(* Logix 5000 project; controller STAT 1756-L72 rev 20.12; software revision 20.04; part 11 of 34 *)
(* tags used below, declared in another part *)
   ai_flow_L1 : REAL;
   ai_flow_L2 : REAL;
   ai_flow_L3 : REAL;
   aux2_P1 : BOOL;
   AUX2_P2 : BOOL;
   aux_P1_ETANG : BOOL;
   AUX_P2 : BOOL;
   AUX_P5_RINC : BOOL;
   B10 : DINT[20];
   B14 : DINT[30];
   B16 : DINT[30];
   B17 : DINT[30];
   B3 : DINT[256];
   B9 : DINT[40];
   EAU_VILLE : BOOL;
   F8 : REAL[256];
   I19_000_Bit14 : ALIAS FOR I19[0].14;   // vanne eau ville open
   I19_000_Bit15 : ALIAS FOR I19[0].15;   // vanne eau ville closed
   I19_001_Bit00 : ALIAS FOR I19[1].0;   // pulse eau de ville
   I1_005_Bit15 : ALIAS FOR I1[5].15;
   I1_008_Bit01 : ALIAS FOR I1[8].1;   // Hand Automaat stormbekken
   I1_008_Bit02 : ALIAS FOR I1[8].2;   // Start pomp 1 stormbekken
   I1_008_Bit03 : ALIAS FOR I1[8].3;   // Stop pomp 1 stormbekken
   I1_008_Bit04 : ALIAS FOR I1[8].4;   // Start pomp 2 stormbekken
   I1_008_Bit05 : ALIAS FOR I1[8].5;   // Stop pomp 2 stormbekken
   I1_008_Bit06 : ALIAS FOR I1[8].6;   // Start P3 stormbekken
   I1_008_Bit07 : ALIAS FOR I1[8].7;   // Stop P3 stormbekken
   I1_008_Bit08 : ALIAS FOR I1[8].8;   // Start PD1 Biocide
   I1_008_Bit09 : ALIAS FOR I1[8].9;   // Stop PD1 biocide
   I1_008_Bit10 : ALIAS FOR I1[8].10;   // start pd2 biocide
   I1_008_Bit11 : ALIAS FOR I1[8].11;   // stop pd2 biocide
   I1_009_Bit05 : ALIAS FOR I1[9].5;   // Pomp 1 in driehoek
   I1_009_Bit06 : ALIAS FOR I1[9].6;   // Pomp 1 in ster
   I1_009_Bit09 : ALIAS FOR I1[9].9;   // Pomp 2 in driehoek
   I1_009_Bit10 : ALIAS FOR I1[9].10;   // Pomp 2 in ster
   I1_009_Bit13 : ALIAS FOR I1[9].13;   // Pomp 3 in driehoek
   I1_009_Bit14 : ALIAS FOR I1[9].14;   // Pomp 3 in ster
   I1_010_Bit05 : ALIAS FOR I1[10].5;   // Vlotterschak lal stormbekken
   I1_010_Bit07 : ALIAS FOR I1[10].7;   // Inpuls promag 33 debiet
   I1_010_Bit10 : ALIAS FOR I1[10].10;   // Noodstop relais ok stormbekken
   I26_000 : ALIAS FOR I26[0];
   I26_003 : ALIAS FOR I26[3];
   I26_004 : ALIAS FOR I26[4];
   I26_005 : ALIAS FOR I26[5];
   I26_007 : ALIAS FOR I26[7];
   I28_000 : ALIAS FOR I28[0];
   I28_001 : ALIAS FOR I28[1];
   I28_002 : ALIAS FOR I28[2];
   I2_000_Bit04 : ALIAS FOR I2[0].4;   // Deelnoodstop cl6 eurowater
   I2_000_Bit05 : ALIAS FOR I2[0].5;   // Deelnoodstop cl7 IBT A
   I4_000_Bit02 : ALIAS FOR I4[0].2;   // defaut drive P4
   I5_001_Bit12 : ALIAS FOR I5[1].12;   // EV6_OPEN
   I5_001_Bit13 : ALIAS FOR I5[1].13;   // EV6_TOE
   I5_001_Bit14 : ALIAS FOR I5[1].14;   // EV7_TOE
   I6_000_Bit00 : ALIAS FOR I6[0].0;   // totaal debiet tfb1
   I6_000_Bit01 : ALIAS FOR I6[0].1;   // totaal debiet stfa 2
   I6_000_Bit07 : ALIAS FOR I6[0].7;   // pulsteller debiet ontijzer 2
   I6_000_Bit15 : ALIAS FOR I6[0].15;   // Lus 1 niveau reservoir kontakt 3
   I6_001_Bit00 : ALIAS FOR I6[1].0;   // hoog alarm ketel pretraitec water
   I6_001_Bit01 : ALIAS FOR I6[1].1;   // Lus 1 niveau ketel hoog
   I6_001_Bit02 : ALIAS FOR I6[1].2;   // laag alarm pretraitec water
   I6_001_Bit03 : ALIAS FOR I6[1].3;   // zeer laag alarm pretraitec water
   I6_001_Bit05 : ALIAS FOR I6[1].5;   // debietsmeting q2 pulsen
   I6_001_Bit08 : ALIAS FOR I6[1].8;   // debietsmeting q3 pulsen
   I7_000_Bit07 : ALIAS FOR I7[0].7;   // hoog alarm ketel tampon
   I7_001_Bit07 : ALIAS FOR I7[1].7;   // q4 inpulsen osmose globaal
   I8_000_Bit04 : ALIAS FOR I8[0].4;   // niveau kuip 20m hoog alarm
   I8_001_Bit09 : ALIAS FOR I8[1].9;   // Schakelaar hand autom cl6
   I9_000_Bit06 : ALIAS FOR I9[0].6;   // Drukknop start CL6 S1
   I9_000_Bit07 : ALIAS FOR I9[0].7;   // Drukknop stop CL6 S1
   I9_000_Bit09 : ALIAS FOR I9[0].9;   // Hand_Auto CL7
   I9_000_Bit10 : ALIAS FOR I9[0].10;   // Drukknop start CL7 P3
   I9_000_Bit11 : ALIAS FOR I9[0].11;   // Drukknop stop CL7 P3
   I9_000_Bit14 : ALIAS FOR I9[0].14;   // Drukknop start CL7 P5
   I9_000_Bit15 : ALIAS FOR I9[0].15;   // Drukknop stop CL7 P5
   ibtlancy1 : DINT;
   KRK_K2 : DINT;
   L1_stat : DINT[20];
   LDN_L2 : REAL;
   LDN_L3 : REAL;
   mem1 : REAL;
   mem3 : REAL;
   mem_water_flow_to_l1 : REAL;
   mem_water_flow_to_l2 : REAL;
   mem_water_flow_to_l31 : REAL;
   MW : BOOL;
   N11 : DINT[150];
   N12 : DINT[230];
   N12_219 : REAL;
   N12_220 : REAL;
   N12_221 : REAL;
   N13 : DINT[230];
   N24 : DINT[80];
   O13_001_Bit13 : ALIAS FOR O13[1].13;   // vanne eau de ville
   O15_001_Bit10 : ALIAS FOR O15[1].10;   // EV6 EV6
   O1_011_Bit00 : ALIAS FOR O1[11].0;
   O1_011_Bit01 : ALIAS FOR O1[11].1;
   O1_011_Bit02 : ALIAS FOR O1[11].2;
   O1_011_Bit03 : ALIAS FOR O1[11].3;
   O1_011_Bit04 : ALIAS FOR O1[11].4;
   O1_011_Bit05 : ALIAS FOR O1[11].5;
   O1_011_Bit06 : ALIAS FOR O1[11].6;
   O1_011_Bit07 : ALIAS FOR O1[11].7;
   O1_011_Bit08 : ALIAS FOR O1[11].8;
   O1_011_Bit09 : ALIAS FOR O1[11].9;
   O1_011_Bit10 : ALIAS FOR O1[11].10;
   ons7 : BOOL;
   ons8 : BOOL;
   ons9 : BOOL;
   P1_ETANG : BOOL;
   P2_ETANG : BOOL;
   P3 : BOOL;
   P4 : BOOL;
   P5_regen : BOOL;
   PRES_LIGNE : REAL;
   QUAT_Q2 : REAL;
   S1 : BOOL;
   s_bp_wissel_P2_usi_tfb : BOOL;   // choix p2 etang vers tfb (1) ou usine (0)
   S_LVL_VIJVER : REAL;
   scp_KRK2 : SCP;
   scp_l1_flow : SCP;
   scp_l2_flow : SCP;
   scp_l3_flow : SCP;
   scp_LDN_2 : SCP;
   scp_LDN_3 : SCP;
   scp_N12_219 : SCP;
   scp_N12_220 : SCP;
   scp_N12_221 : SCP;
   scp_PRES_LIGNE : SCP;
   scp_quat_2 : SCP;
   t1min : TIMER;
   T27 : TIMER[100];
   T4 : TIMER[200];
   water_flow_to_l1 : REAL;
   water_flow_to_l1_inst : REAL;
   water_flow_to_l2 : REAL;
   water_flow_to_l2_inst : REAL;
   water_flow_to_l3 : REAL;
   water_flow_to_l3_inst1 : REAL;
(* ibt, continued *)

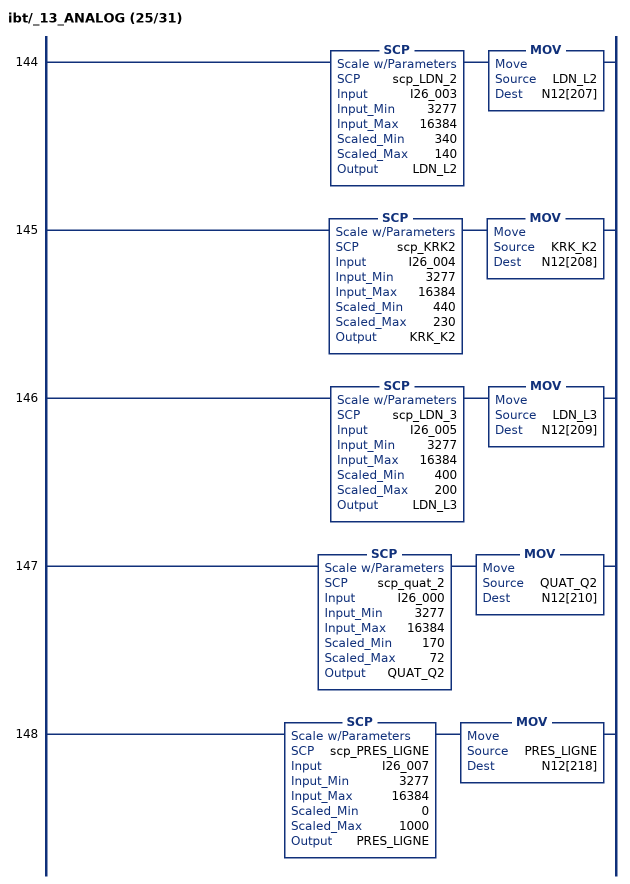
   [picture p154: ibt/_13_ANALOG rungs 144-148]
   144: SCP(scp_LDN_2,I26_003,3277,16384,340,140,LDN_L2)MOV(LDN_L2,N12[207]);
   145: SCP(scp_KRK2,I26_004,3277,16384,440,230,KRK_K2)MOV(KRK_K2,N12[208]);
   146: SCP(scp_LDN_3,I26_005,3277,16384,400,200,LDN_L3)MOV(LDN_L3,N12[209]);
   147: SCP(scp_quat_2,I26_000,3277,16384,170,72,QUAT_Q2)MOV(QUAT_Q2,N12[210]);
   148: SCP(scp_PRES_LIGNE,I26_007,3277,16384,0,1000,PRES_LIGNE)MOV(PRES_LIGNE,N12[218]);
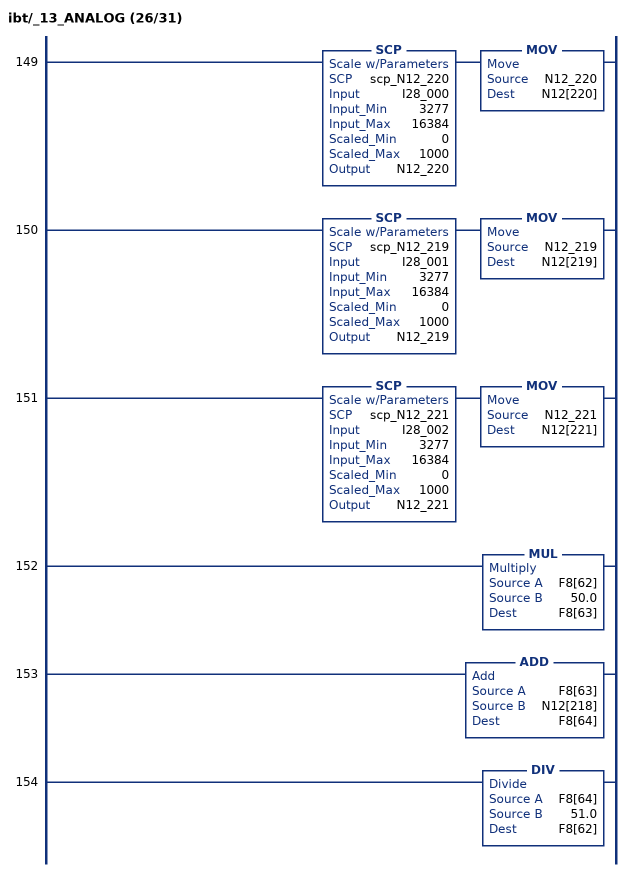
   149: SCP(scp_N12_220,I28_000,3277,16384,0,1000,N12_220)MOV(N12_220,N12[220]);
   150: SCP(scp_N12_219,I28_001,3277,16384,0,1000,N12_219)MOV(N12_219,N12[219]);
   151: SCP(scp_N12_221,I28_002,3277,16384,0,1000,N12_221)MOV(N12_221,N12[221]);
   152: MUL(F8[62],50.0,F8[63]);
   153: ADD(F8[63],N12[218],F8[64]);
   154: DIV(F8[64],51.0,F8[62]);
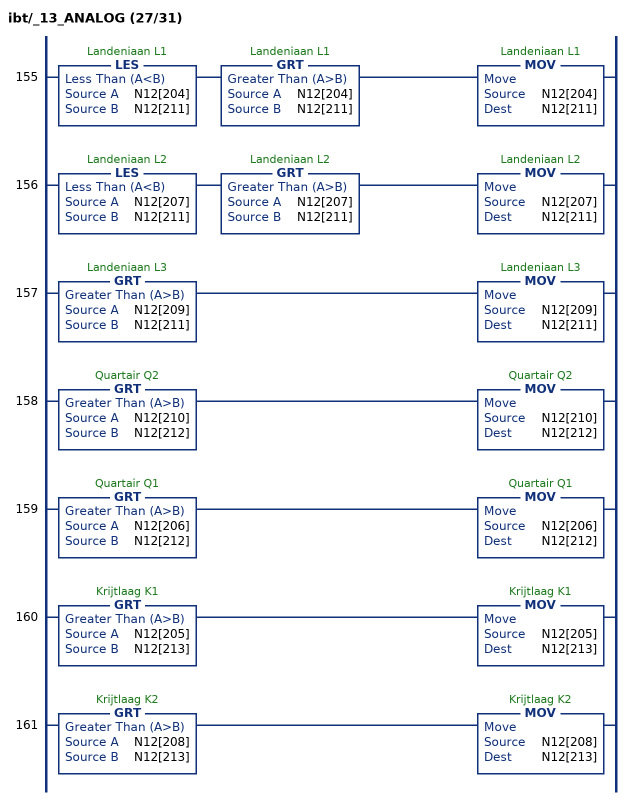
   155: LES(N12[204],N12[211])GRT(N12[204],N12[211])MOV(N12[204],N12[211]);
   156: LES(N12[207],N12[211])GRT(N12[207],N12[211])MOV(N12[207],N12[211]);
   157: GRT(N12[209],N12[211])MOV(N12[209],N12[211]);
   158: GRT(N12[210],N12[212])MOV(N12[210],N12[212]);
   159: GRT(N12[206],N12[212])MOV(N12[206],N12[212]);
   160: GRT(N12[205],N12[213])MOV(N12[205],N12[213]);
   161: GRT(N12[208],N12[213])MOV(N12[208],N12[213]);
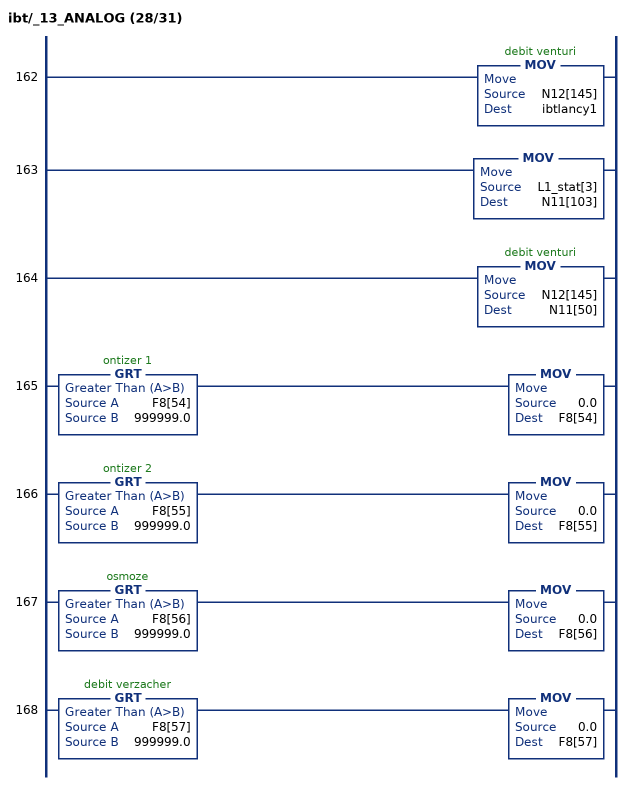
   162: MOV(N12[145],ibtlancy1);
   163: MOV(L1_stat[3],N11[103]);
   164: MOV(N12[145],N11[50]);
   165: GRT(F8[54],999999.0)MOV(0.0,F8[54]);
   166: GRT(F8[55],999999.0)MOV(0.0,F8[55]);
   167: GRT(F8[56],999999.0)MOV(0.0,F8[56]);
   168: GRT(F8[57],999999.0)MOV(0.0,F8[57]);
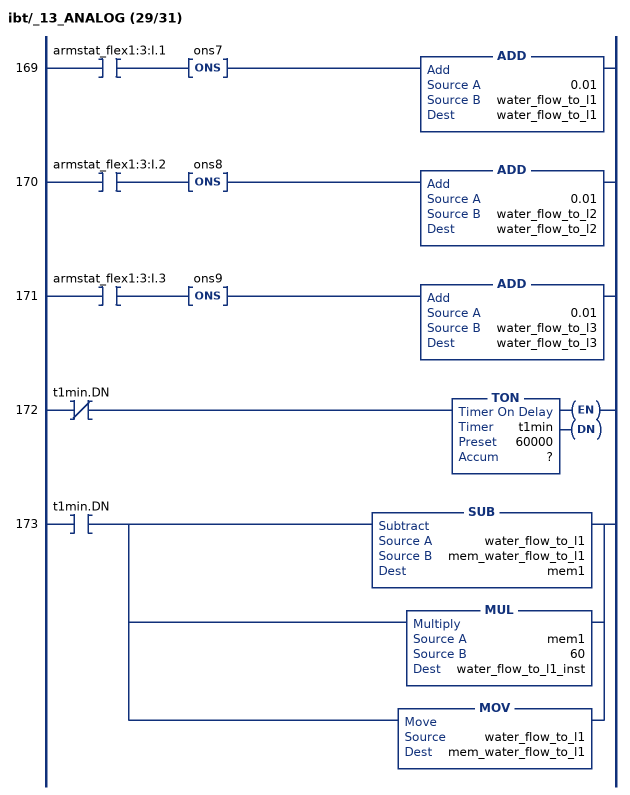
   169: XIC(armstat_flex1:3:I.1)ONS(ons7)ADD(0.01,water_flow_to_l1,water_flow_to_l1);
   170: XIC(armstat_flex1:3:I.2)ONS(ons8)ADD(0.01,water_flow_to_l2,water_flow_to_l2);
   171: XIC(armstat_flex1:3:I.3)ONS(ons9)ADD(0.01,water_flow_to_l3,water_flow_to_l3);
   172: XIO(t1min.DN)TON(t1min,?,?);
   173: XIC(t1min.DN)[SUB(water_flow_to_l1,mem_water_flow_to_l1,mem1) ,MUL(mem1,60,water_flow_to_l1_inst) ,MOV(water_flow_to_l1,mem_water_flow_to_l1) ];
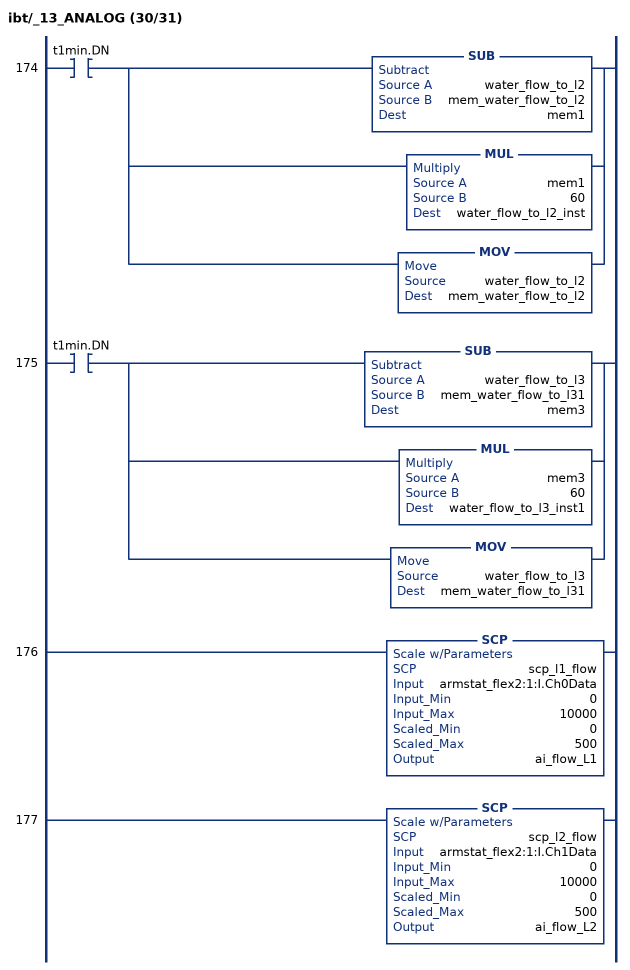
   174: XIC(t1min.DN)[SUB(water_flow_to_l2,mem_water_flow_to_l2,mem1) ,MUL(mem1,60,water_flow_to_l2_inst) ,MOV(water_flow_to_l2,mem_water_flow_to_l2) ];
   175: XIC(t1min.DN)[SUB(water_flow_to_l3,mem_water_flow_to_l31,mem3) ,MUL(mem3,60,water_flow_to_l3_inst1) ,MOV(water_flow_to_l3,mem_water_flow_to_l31) ];
   176: SCP(scp_l1_flow,armstat_flex2:1:I.Ch0Data,0,10000,0,500,ai_flow_L1);
   177: SCP(scp_l2_flow,armstat_flex2:1:I.Ch1Data,0,10000,0,500,ai_flow_L2);
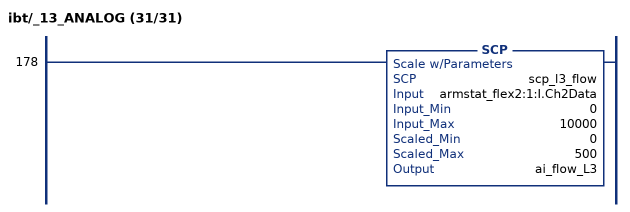
   178: SCP(scp_l3_flow,armstat_flex2:1:I.Ch2Data,0,10000,0,500,ai_flow_L3);
END_ROUTINE

ROUTINE _14_P1_P5_PD1   (* ladder *)
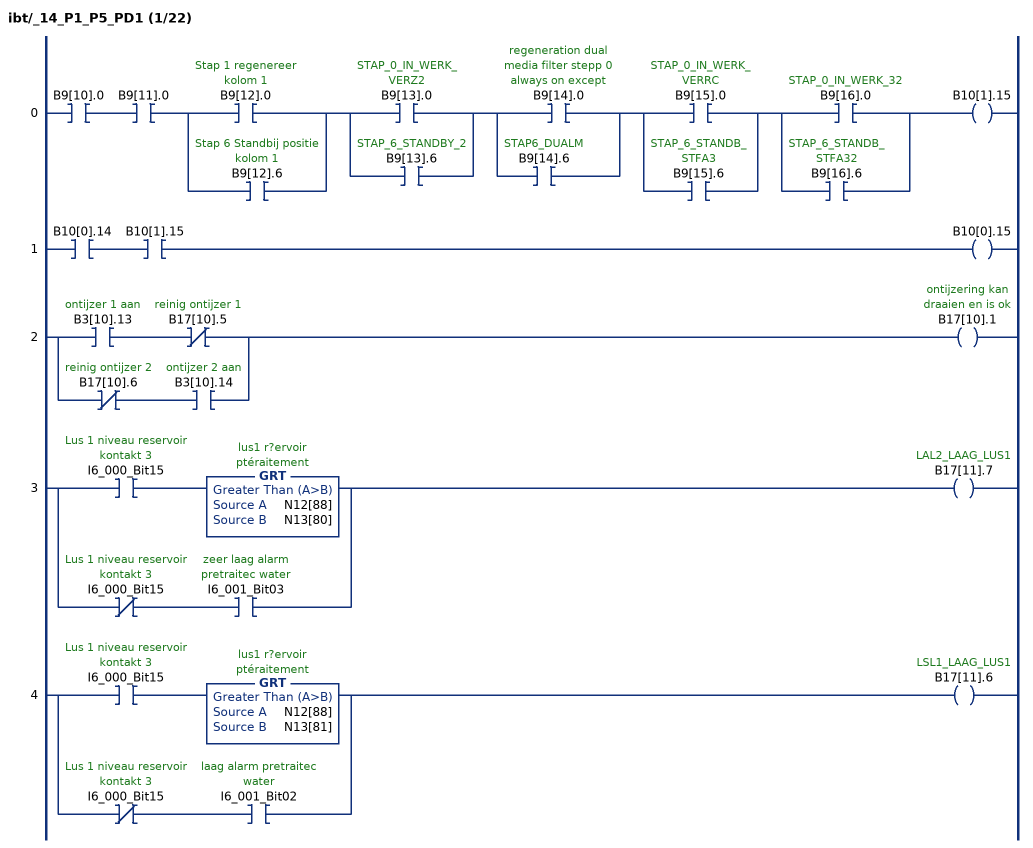
   0: XIC(B9[10].0)XIC(B9[11].0)[XIC(B9[12].0) ,XIC(B9[12].6) ][XIC(B9[13].0) ,XIC(B9[13].6) ][XIC(B9[14].0) ,XIC(B9[14].6) ][XIC(B9[15].0) ,XIC(B9[15].6) ][XIC(B9[16].0) ,XIC(B9[16].6) ]OTE(B10[1].15);
   1: XIC(B10[0].14)XIC(B10[1].15)OTE(B10[0].15);
   2: [XIC(B3[10].13) XIO(B17[10].5) ,XIO(B17[10].6) XIC(B3[10].14) ]OTE(B17[10].1);
   3: [XIC(I6_000_Bit15) GRT(N12[88],N13[80]) ,XIO(I6_000_Bit15) XIC(I6_001_Bit03) ]OTE(B17[11].7);
   4: [XIC(I6_000_Bit15) GRT(N12[88],N13[81]) ,XIO(I6_000_Bit15) XIC(I6_001_Bit02) ]OTE(B17[11].6);
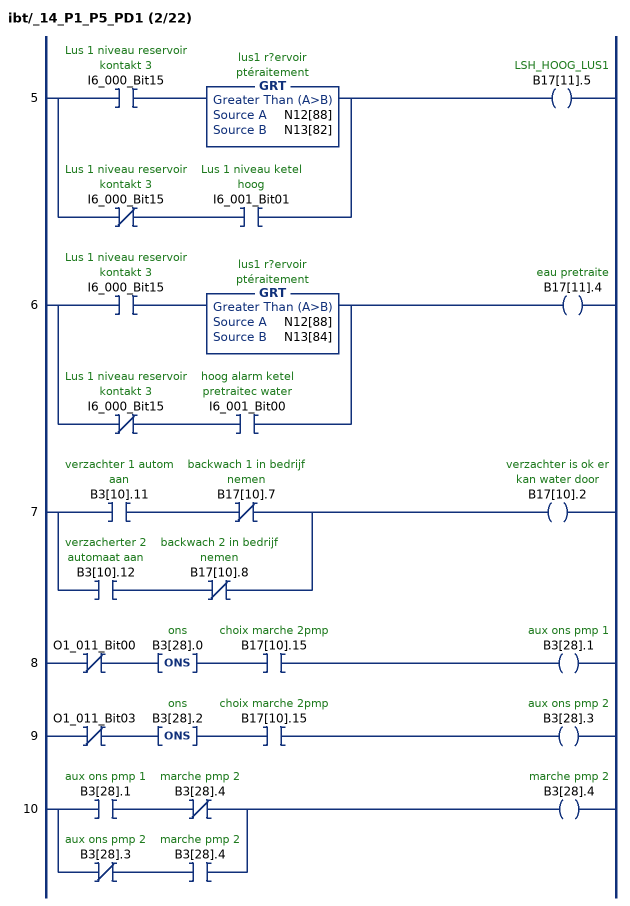
   5: [XIC(I6_000_Bit15) GRT(N12[88],N13[82]) ,XIO(I6_000_Bit15) XIC(I6_001_Bit01) ]OTE(B17[11].5);
   6: [XIC(I6_000_Bit15) GRT(N12[88],N13[84]) ,XIO(I6_000_Bit15) XIC(I6_001_Bit00) ]OTE(B17[11].4);
   7: [XIC(B3[10].11) XIO(B17[10].7) ,XIC(B3[10].12) XIO(B17[10].8) ]OTE(B17[10].2);
   8: XIO(O1_011_Bit00)ONS(B3[28].0)XIC(B17[10].15)OTE(B3[28].1);
   9: XIO(O1_011_Bit03)ONS(B3[28].2)XIC(B17[10].15)OTE(B3[28].3);
   10: [XIC(B3[28].1) XIO(B3[28].4) ,XIO(B3[28].3) XIC(B3[28].4) ]OTE(B3[28].4);
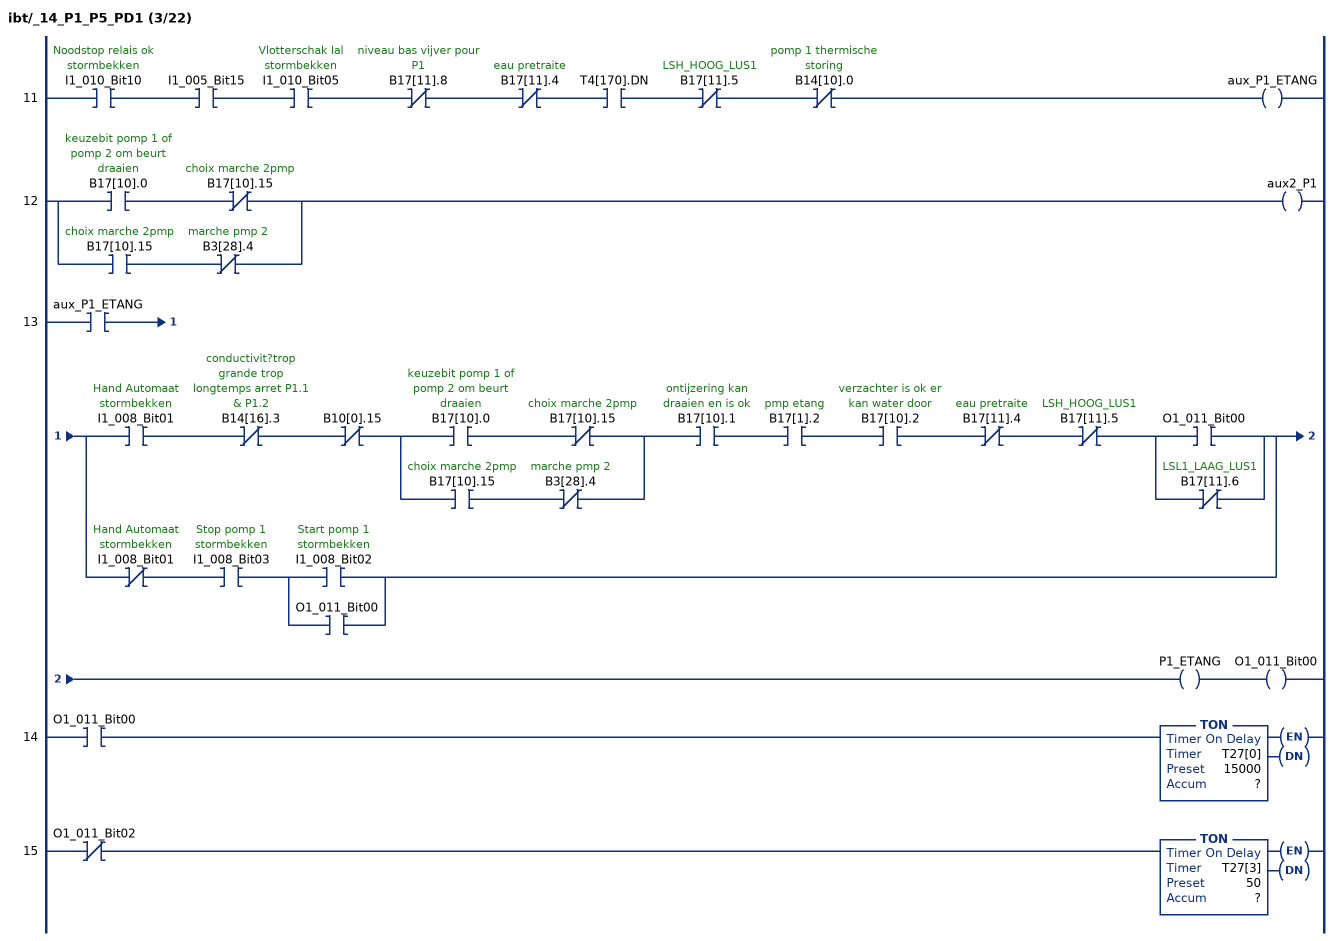
   11: XIC(I1_010_Bit10)XIC(I1_005_Bit15)XIC(I1_010_Bit05)XIO(B17[11].8)XIO(B17[11].4)XIC(T4[170].DN)XIO(B17[11].5)XIO(B14[10].0)OTE(aux_P1_ETANG);
   12: [XIC(B17[10].0) XIO(B17[10].15) ,XIC(B17[10].15) XIO(B3[28].4) ]OTE(aux2_P1);
   13: XIC(aux_P1_ETANG)[XIC(I1_008_Bit01) XIO(B14[16].3) XIO(B10[0].15) [XIC(B17[10].0) XIO(B17[10].15) ,XIC(B17[10].15) XIO(B3[28].4) ] XIC(B17[10].1) XIC(B17[1].2) XIC(B17[10].2) XIO(B17[11].4) XIO(B17[11].5) [XIC(O1_011_Bit00) ,XIO(B17[11].6) ] ,XIO(I1_008_Bit01) XIC(I1_008_Bit03) [XIC(I1_008_Bit02) ,XIC(O1_011_Bit00) ] ]OTE(P1_ETANG)OTE(O1_011_Bit00);
   14: XIC(O1_011_Bit00)TON(T27[0],?,?);
   15: XIO(O1_011_Bit02)TON(T27[3],?,?);
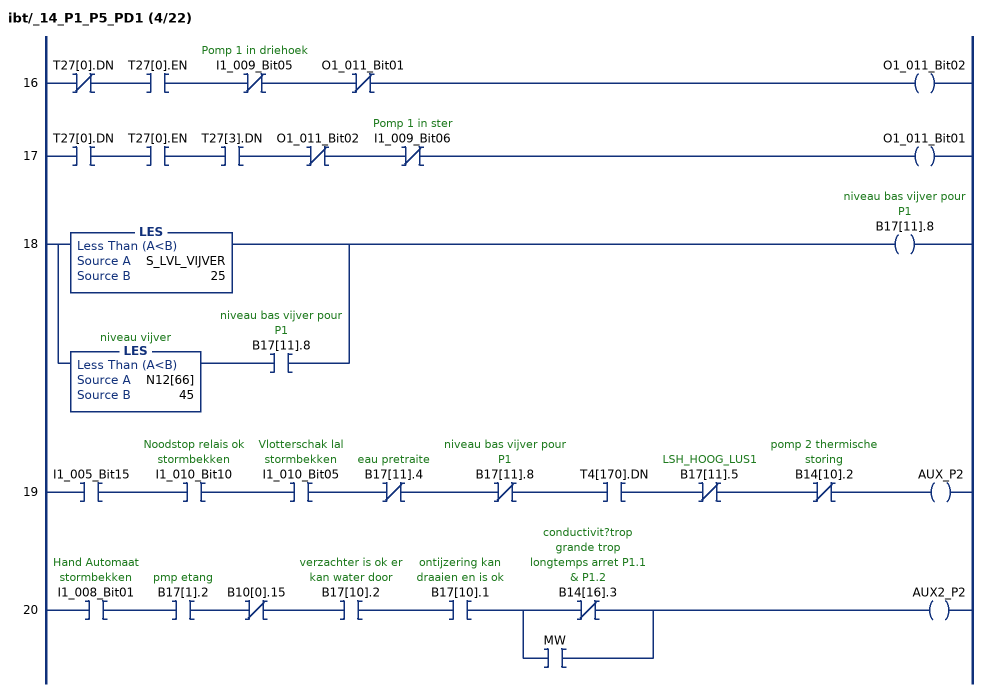
   16: XIO(T27[0].DN)XIC(T27[0].EN)XIO(I1_009_Bit05)XIO(O1_011_Bit01)OTE(O1_011_Bit02);
   17: XIC(T27[0].DN)XIC(T27[0].EN)XIC(T27[3].DN)XIO(O1_011_Bit02)XIO(I1_009_Bit06)OTE(O1_011_Bit01);
   18: [LES(S_LVL_VIJVER,25) ,LES(N12[66],45) XIC(B17[11].8) ]OTE(B17[11].8);
   19: XIC(I1_005_Bit15)XIC(I1_010_Bit10)XIC(I1_010_Bit05)XIO(B17[11].4)XIO(B17[11].8)XIC(T4[170].DN)XIO(B17[11].5)XIO(B14[10].2)OTE(AUX_P2);
   20: XIC(I1_008_Bit01)XIC(B17[1].2)XIO(B10[0].15)XIC(B17[10].2)XIC(B17[10].1)[XIO(B14[16].3) ,XIC(MW) ]OTE(AUX2_P2);
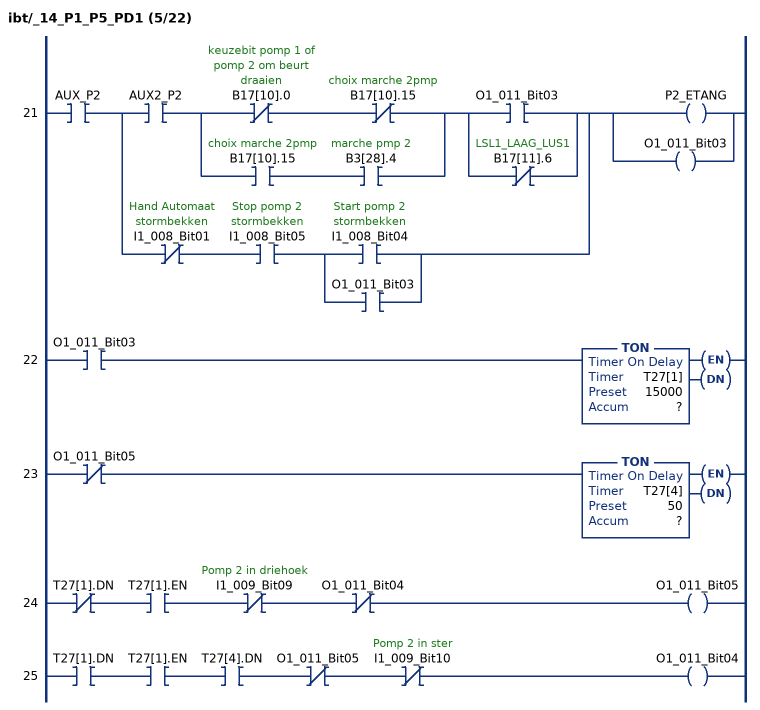
   21: XIC(AUX_P2)[XIC(AUX2_P2) [XIO(B17[10].0) XIO(B17[10].15) ,XIC(B17[10].15) XIC(B3[28].4) ] [XIC(O1_011_Bit03) ,XIO(B17[11].6) ] ,XIO(I1_008_Bit01) XIC(I1_008_Bit05) [XIC(I1_008_Bit04) ,XIC(O1_011_Bit03) ] ][OTE(P2_ETANG) ,OTE(O1_011_Bit03) ];
   22: XIC(O1_011_Bit03)TON(T27[1],?,?);
   23: XIO(O1_011_Bit05)TON(T27[4],?,?);
   24: XIO(T27[1].DN)XIC(T27[1].EN)XIO(I1_009_Bit09)XIO(O1_011_Bit04)OTE(O1_011_Bit05);
   25: XIC(T27[1].DN)XIC(T27[1].EN)XIC(T27[4].DN)XIO(O1_011_Bit05)XIO(I1_009_Bit10)OTE(O1_011_Bit04);
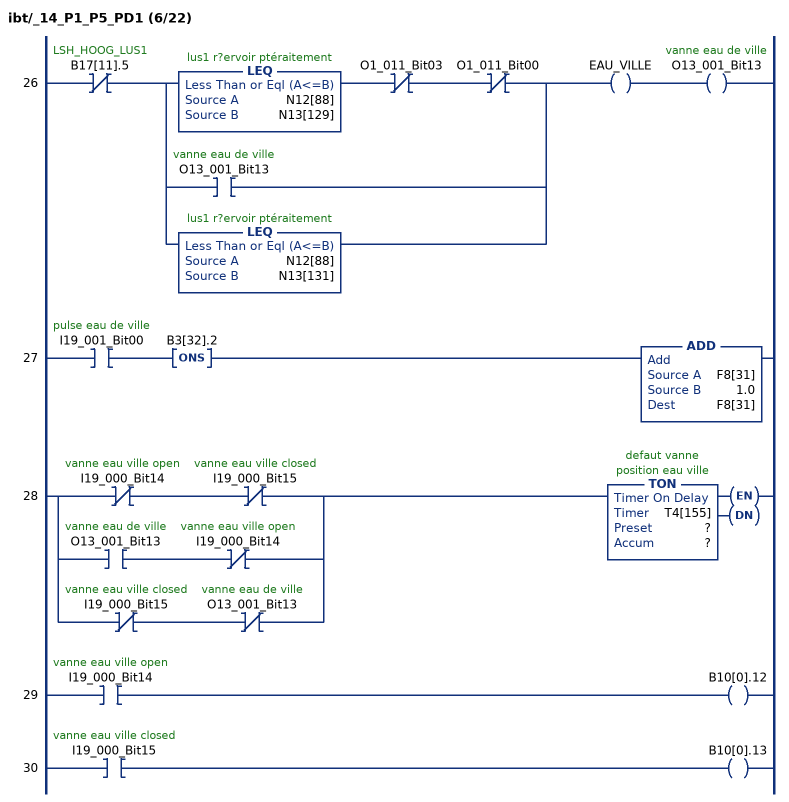
   26: XIO(B17[11].5)[LEQ(N12[88],N13[129]) XIO(O1_011_Bit03) XIO(O1_011_Bit00) ,XIC(O13_001_Bit13) ,LEQ(N12[88],N13[131]) ]OTE(EAU_VILLE)OTE(O13_001_Bit13);
   27: XIC(I19_001_Bit00)ONS(B3[32].2)ADD(F8[31],1.0,F8[31]);
   28: [XIO(I19_000_Bit14) XIO(I19_000_Bit15) ,XIC(O13_001_Bit13) XIO(I19_000_Bit14) ,XIO(I19_000_Bit15) XIO(O13_001_Bit13) ]TON(T4[155],?,?);
   29: XIC(I19_000_Bit14)OTE(B10[0].12);
   30: XIC(I19_000_Bit15)OTE(B10[0].13);
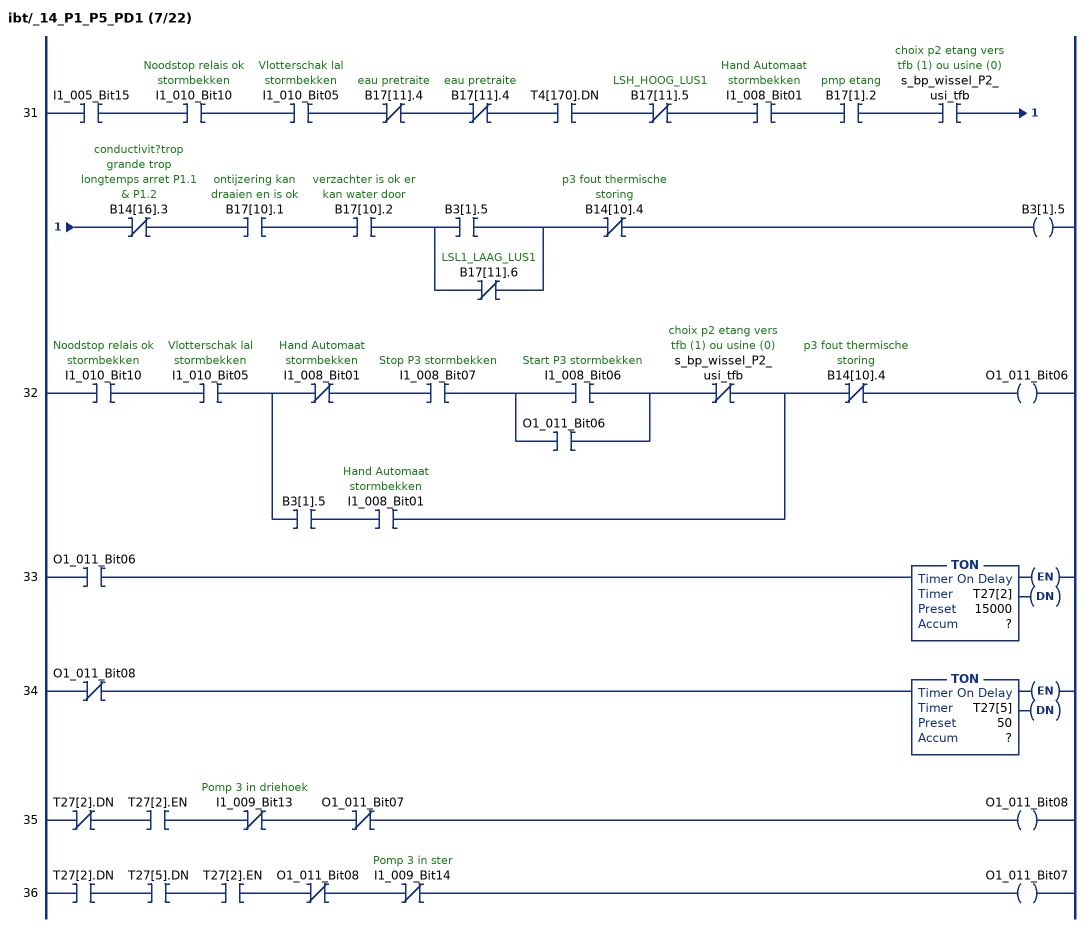
   31: XIC(I1_005_Bit15)XIC(I1_010_Bit10)XIC(I1_010_Bit05)XIO(B17[11].4)XIO(B17[11].4)XIC(T4[170].DN)XIO(B17[11].5)XIC(I1_008_Bit01)XIC(B17[1].2)XIC(s_bp_wissel_P2_usi_tfb)XIO(B14[16].3)XIC(B17[10].1)XIC(B17[10].2)[XIC(B3[1].5) ,XIO(B17[11].6) ]XIO(B14[10].4)OTE(B3[1].5);
   32: XIC(I1_010_Bit10)XIC(I1_010_Bit05)[XIO(I1_008_Bit01) XIC(I1_008_Bit07) [XIC(I1_008_Bit06) ,XIC(O1_011_Bit06) ] XIO(s_bp_wissel_P2_usi_tfb) ,XIC(B3[1].5) XIC(I1_008_Bit01) ]XIO(B14[10].4)OTE(O1_011_Bit06);
   33: XIC(O1_011_Bit06)TON(T27[2],?,?);
   34: XIO(O1_011_Bit08)TON(T27[5],?,?);
   35: XIO(T27[2].DN)XIC(T27[2].EN)XIO(I1_009_Bit13)XIO(O1_011_Bit07)OTE(O1_011_Bit08);
   36: XIC(T27[2].DN)XIC(T27[5].DN)XIC(T27[2].EN)XIO(O1_011_Bit08)XIO(I1_009_Bit14)OTE(O1_011_Bit07);
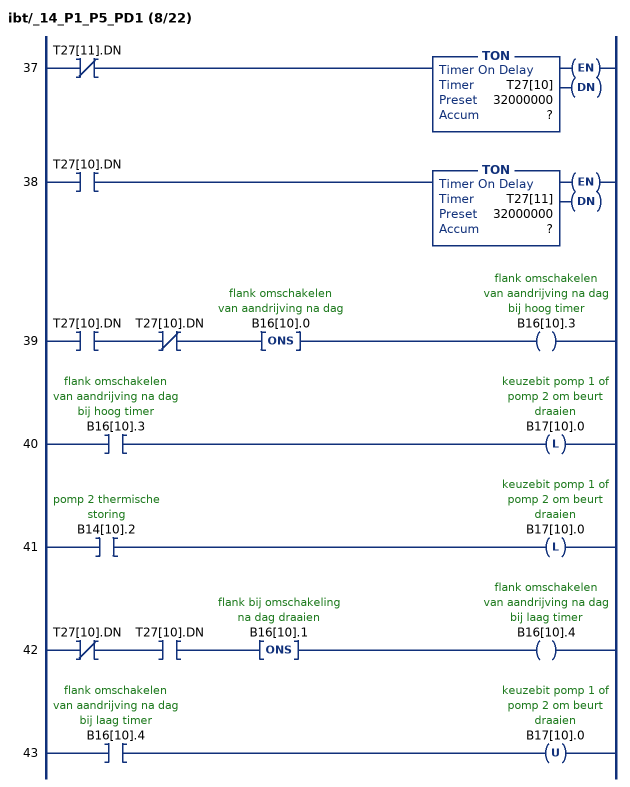
   37: XIO(T27[11].DN)TON(T27[10],?,?);
   38: XIC(T27[10].DN)TON(T27[11],?,?);
   39: XIC(T27[10].DN)XIO(T27[10].DN)ONS(B16[10].0)OTE(B16[10].3);
   40: XIC(B16[10].3)OTL(B17[10].0);
   41: XIC(B14[10].2)OTL(B17[10].0);
   42: XIO(T27[10].DN)XIC(T27[10].DN)ONS(B16[10].1)OTE(B16[10].4);
   43: XIC(B16[10].4)OTU(B17[10].0);
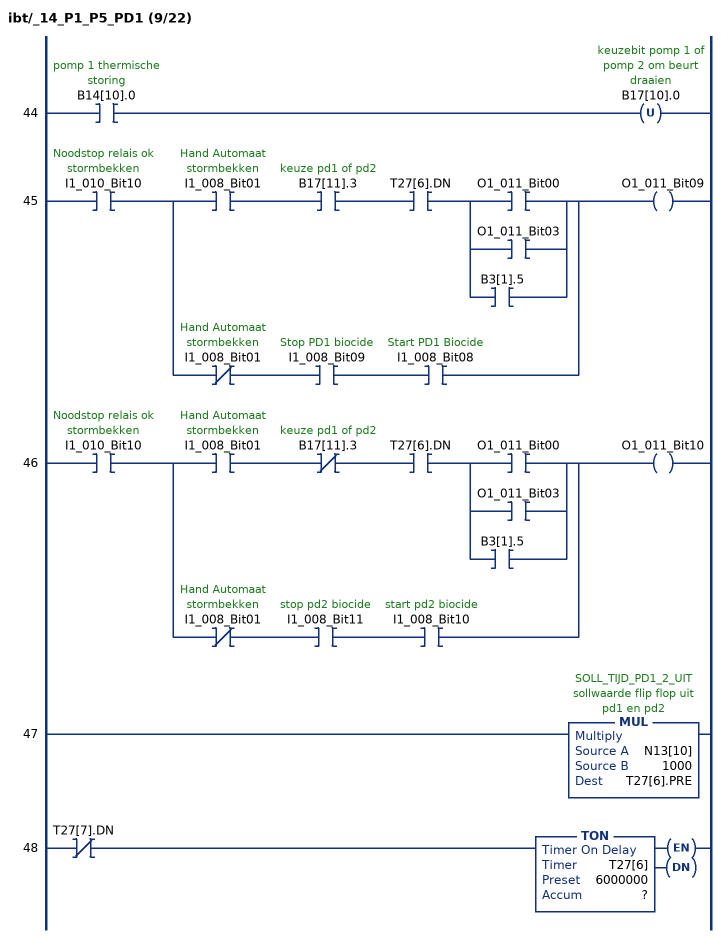
   44: XIC(B14[10].0)OTU(B17[10].0);
   45: XIC(I1_010_Bit10)[XIC(I1_008_Bit01) XIC(B17[11].3) XIC(T27[6].DN) [XIC(O1_011_Bit00) ,XIC(O1_011_Bit03) ,XIC(B3[1].5) ] ,XIO(I1_008_Bit01) XIC(I1_008_Bit09) XIC(I1_008_Bit08) ]OTE(O1_011_Bit09);
   46: XIC(I1_010_Bit10)[XIC(I1_008_Bit01) XIO(B17[11].3) XIC(T27[6].DN) [XIC(O1_011_Bit00) ,XIC(O1_011_Bit03) ,XIC(B3[1].5) ] ,XIO(I1_008_Bit01) XIC(I1_008_Bit11) XIC(I1_008_Bit10) ]OTE(O1_011_Bit10);
   47: MUL(N13[10],1000,T27[6].PRE);
   48: XIO(T27[7].DN)TON(T27[6],?,?);
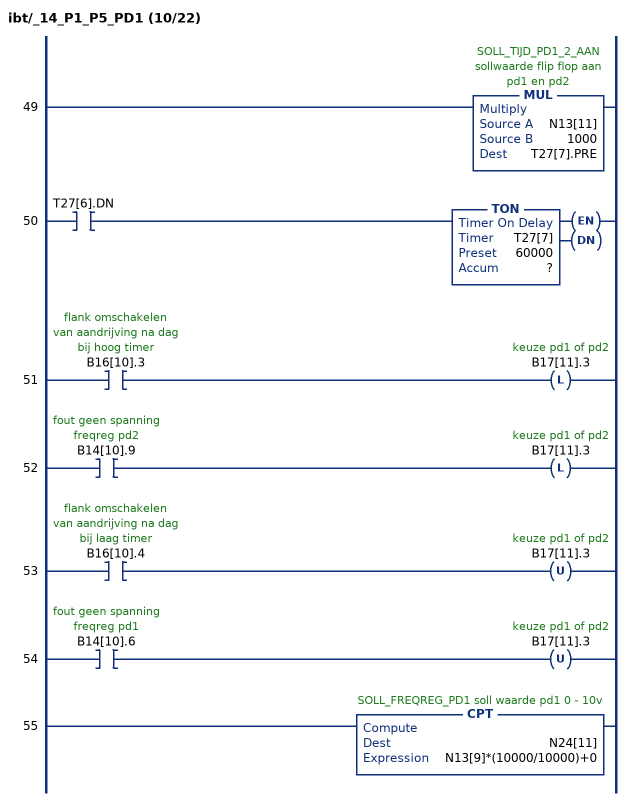
   49: MUL(N13[11],1000,T27[7].PRE);
   50: XIC(T27[6].DN)TON(T27[7],?,?);
   51: XIC(B16[10].3)OTL(B17[11].3);
   52: XIC(B14[10].9)OTL(B17[11].3);
   53: XIC(B16[10].4)OTU(B17[11].3);
   54: XIC(B14[10].6)OTU(B17[11].3);
   55: CPT(N24[11],N13[9]*(10000/10000)+0);
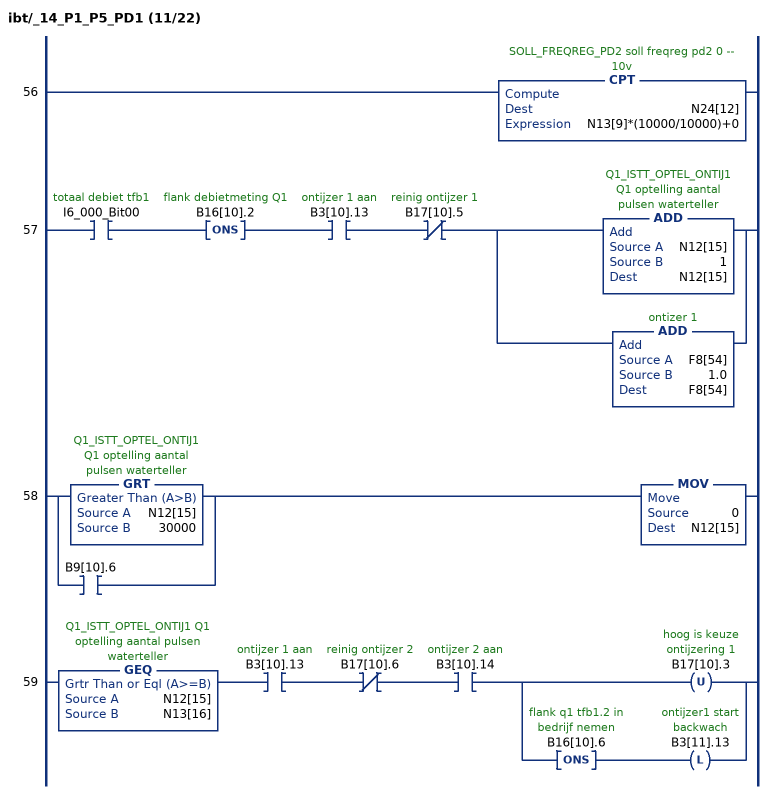
   56: CPT(N24[12],N13[9]*(10000/10000)+0);
   57: XIC(I6_000_Bit00)ONS(B16[10].2)XIC(B3[10].13)XIO(B17[10].5)[ADD(N12[15],1,N12[15]) ,ADD(F8[54],1.0,F8[54]) ];
   58: [GRT(N12[15],30000) ,XIC(B9[10].6) ]MOV(0,N12[15]);
   59: GEQ(N12[15],N13[16])XIC(B3[10].13)XIO(B17[10].6)XIC(B3[10].14)[OTU(B17[10].3) ,ONS(B16[10].6) OTL(B3[11].13) ];
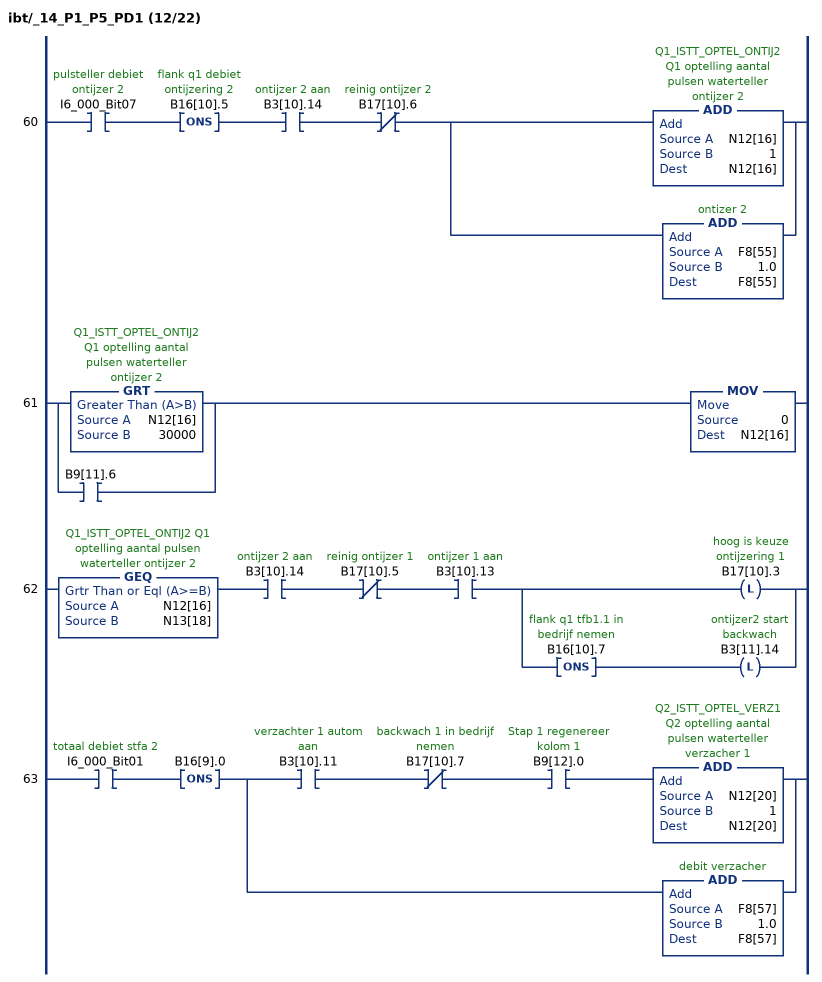
   60: XIC(I6_000_Bit07)ONS(B16[10].5)XIC(B3[10].14)XIO(B17[10].6)[ADD(N12[16],1,N12[16]) ,ADD(F8[55],1.0,F8[55]) ];
   61: [GRT(N12[16],30000) ,XIC(B9[11].6) ]MOV(0,N12[16]);
   62: GEQ(N12[16],N13[18])XIC(B3[10].14)XIO(B17[10].5)XIC(B3[10].13)[OTL(B17[10].3) ,ONS(B16[10].7) OTL(B3[11].14) ];
   63: XIC(I6_000_Bit01)ONS(B16[9].0)[XIC(B3[10].11) XIO(B17[10].7) XIC(B9[12].0) ADD(N12[20],1,N12[20]) ,ADD(F8[57],1.0,F8[57]) ];
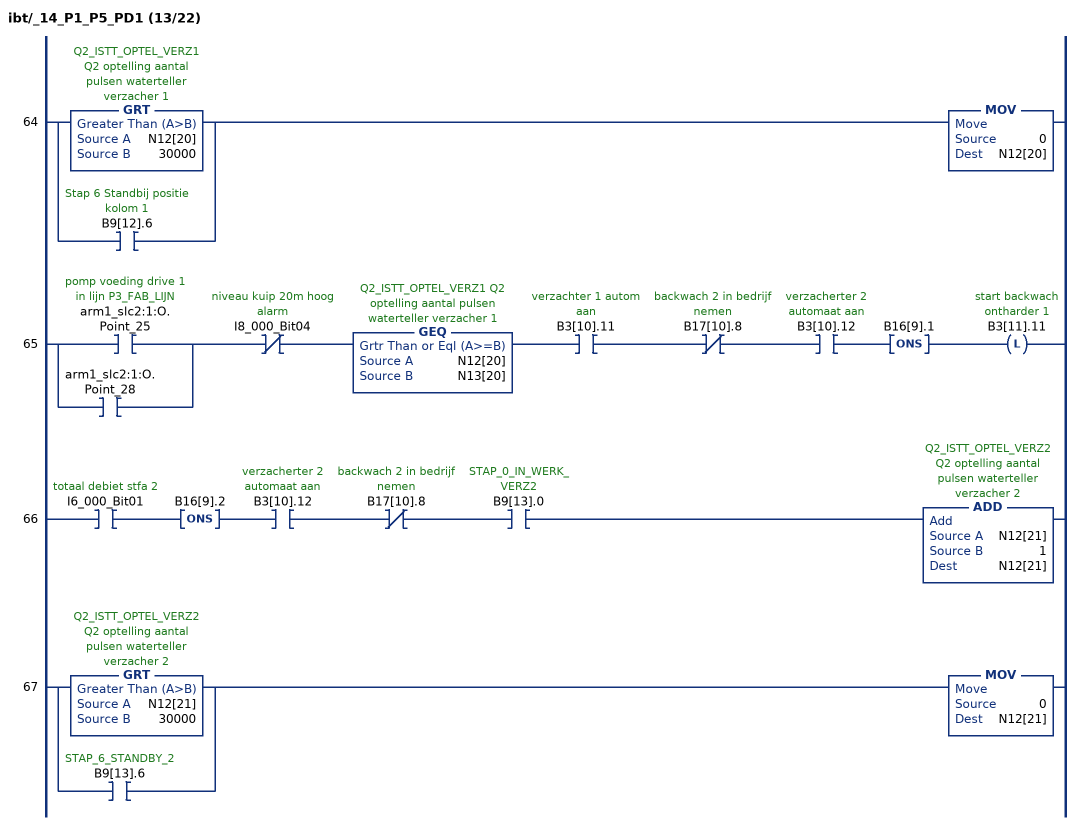
   64: [GRT(N12[20],30000) ,XIC(B9[12].6) ]MOV(0,N12[20]);
   65: [XIC(arm1_slc2:1:O.Point_25) ,XIC(arm1_slc2:1:O.Point_28) ]XIO(I8_000_Bit04)GEQ(N12[20],N13[20])XIC(B3[10].11)XIO(B17[10].8)XIC(B3[10].12)ONS(B16[9].1)OTL(B3[11].11);
   66: XIC(I6_000_Bit01)ONS(B16[9].2)XIC(B3[10].12)XIO(B17[10].8)XIC(B9[13].0)ADD(N12[21],1,N12[21]);
   67: [GRT(N12[21],30000) ,XIC(B9[13].6) ]MOV(0,N12[21]);
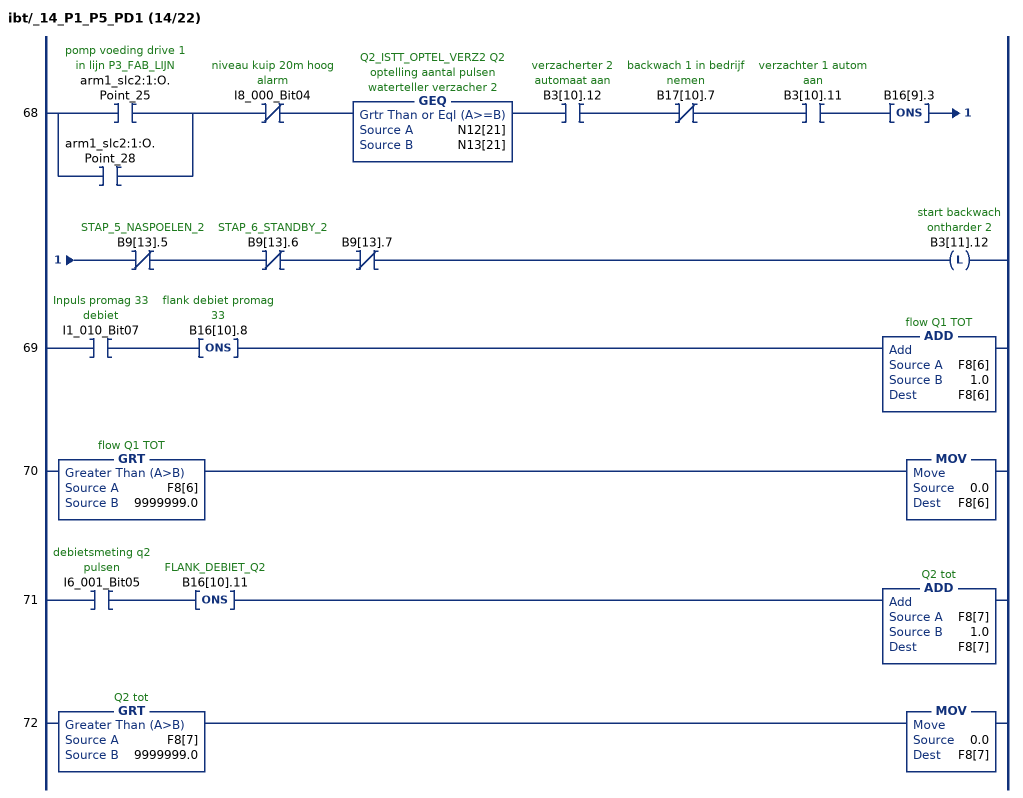
   68: [XIC(arm1_slc2:1:O.Point_25) ,XIC(arm1_slc2:1:O.Point_28) ]XIO(I8_000_Bit04)GEQ(N12[21],N13[21])XIC(B3[10].12)XIO(B17[10].7)XIC(B3[10].11)ONS(B16[9].3)XIO(B9[13].5)XIO(B9[13].6)XIO(B9[13].7)OTL(B3[11].12);
   69: XIC(I1_010_Bit07)ONS(B16[10].8)ADD(F8[6],1.0,F8[6]);
   70: GRT(F8[6],9999999.0)MOV(0.0,F8[6]);
   71: XIC(I6_001_Bit05)ONS(B16[10].11)ADD(F8[7],1.0,F8[7]);
   72: GRT(F8[7],9999999.0)MOV(0.0,F8[7]);
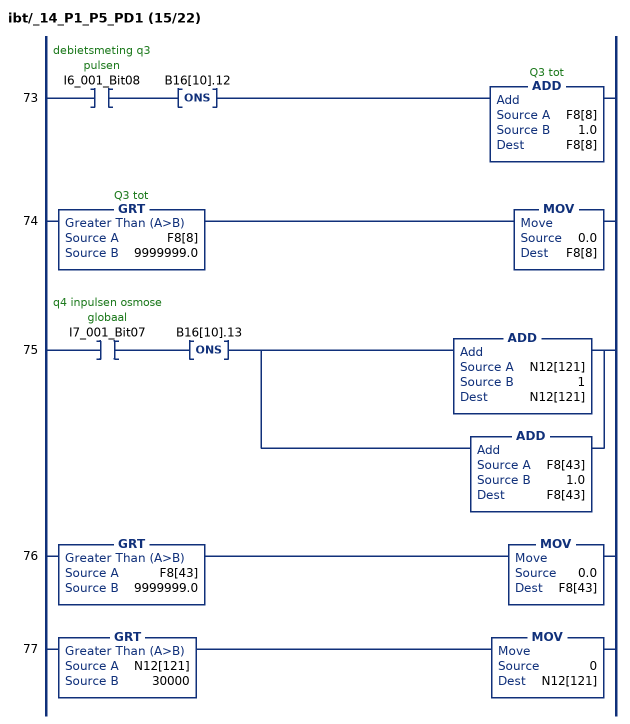
   73: XIC(I6_001_Bit08)ONS(B16[10].12)ADD(F8[8],1.0,F8[8]);
   74: GRT(F8[8],9999999.0)MOV(0.0,F8[8]);
   75: XIC(I7_001_Bit07)ONS(B16[10].13)[ADD(N12[121],1,N12[121]) ,ADD(F8[43],1.0,F8[43]) ];
   76: GRT(F8[43],9999999.0)MOV(0.0,F8[43]);
   77: GRT(N12[121],30000)MOV(0,N12[121]);
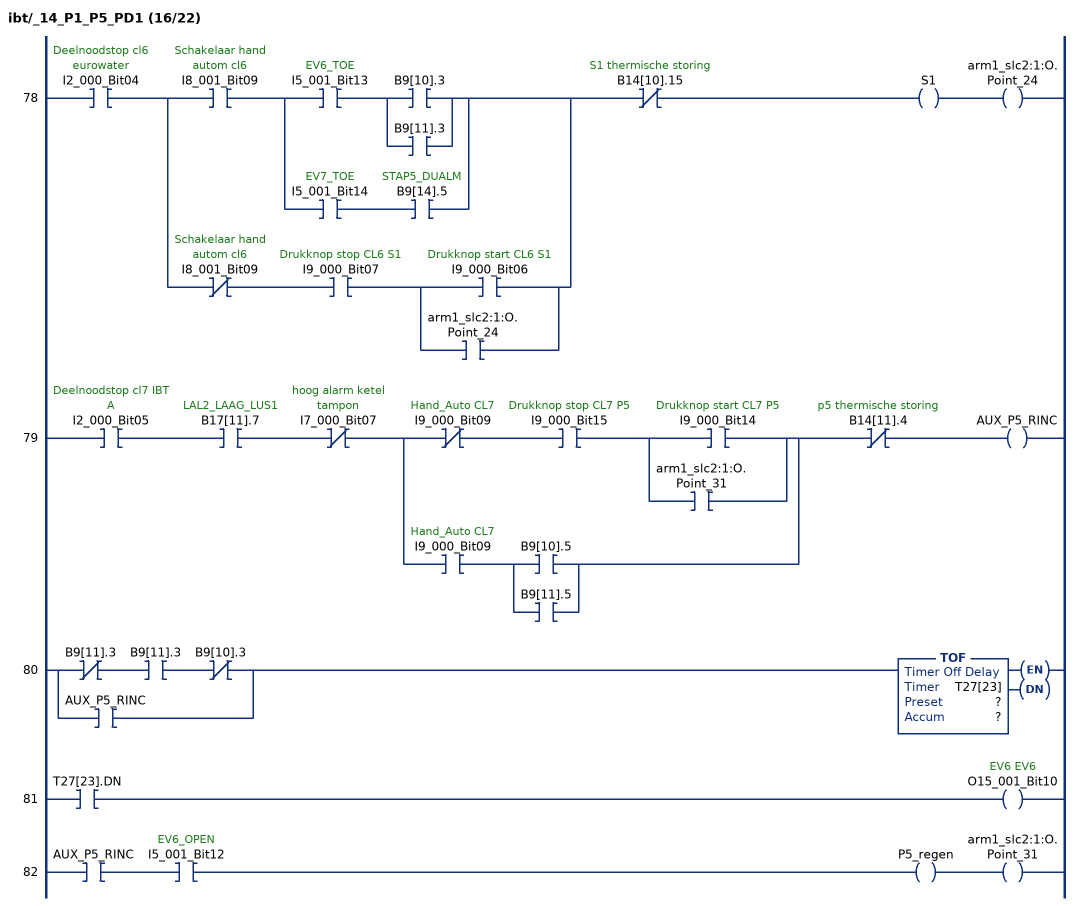
   78: XIC(I2_000_Bit04)[XIC(I8_001_Bit09) [XIC(I5_001_Bit13) [XIC(B9[10].3) ,XIC(B9[11].3) ] ,XIC(I5_001_Bit14) XIC(B9[14].5) ] ,XIO(I8_001_Bit09) XIC(I9_000_Bit07) [XIC(I9_000_Bit06) ,XIC(arm1_slc2:1:O.Point_24) ] ]XIO(B14[10].15)OTE(S1)OTE(arm1_slc2:1:O.Point_24);
   79: XIC(I2_000_Bit05)XIC(B17[11].7)XIO(I7_000_Bit07)[XIO(I9_000_Bit09) XIC(I9_000_Bit15) [XIC(I9_000_Bit14) ,XIC(arm1_slc2:1:O.Point_31) ] ,XIC(I9_000_Bit09) [XIC(B9[10].5) ,XIC(B9[11].5) ] ]XIO(B14[11].4)OTE(AUX_P5_RINC);
   80: [XIO(B9[11].3) XIC(B9[11].3) XIO(B9[10].3) ,XIC(AUX_P5_RINC) ]TOF(T27[23],?,?);
   81: XIC(T27[23].DN)OTE(O15_001_Bit10);
   82: XIC(AUX_P5_RINC)XIC(I5_001_Bit12)OTE(P5_regen)OTE(arm1_slc2:1:O.Point_31);
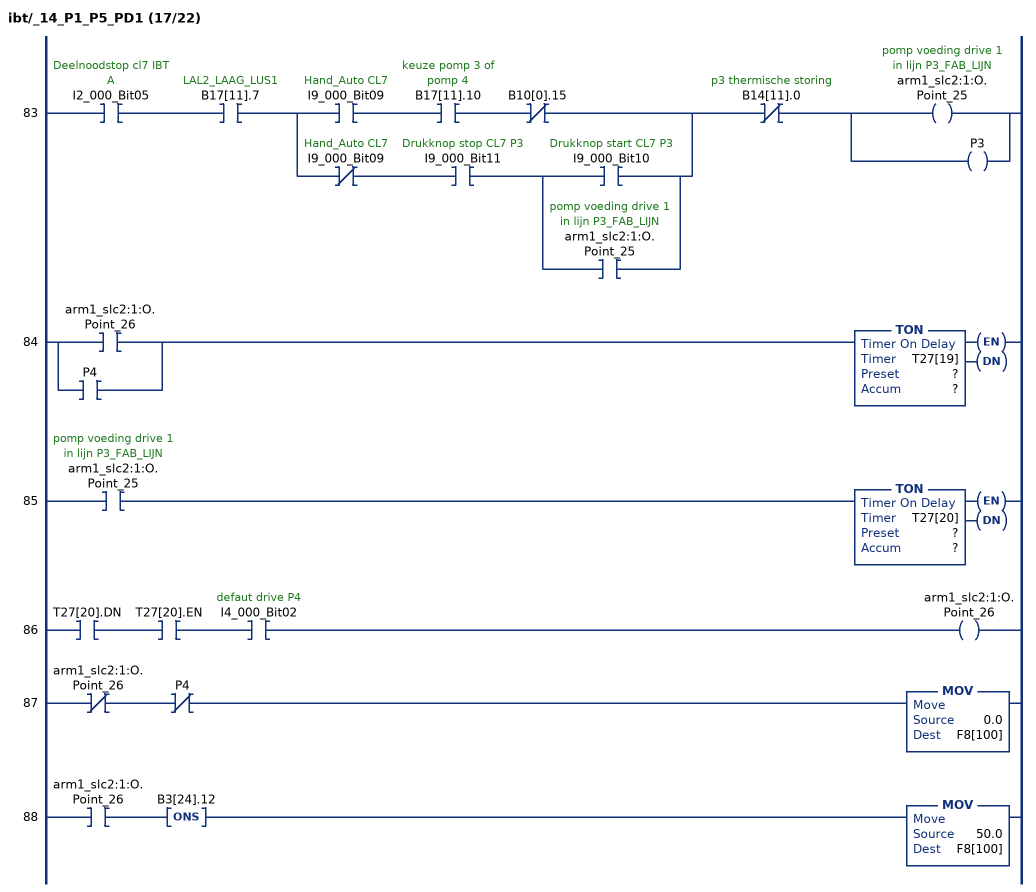
   83: XIC(I2_000_Bit05)XIC(B17[11].7)[XIC(I9_000_Bit09) XIC(B17[11].10) XIO(B10[0].15) ,XIO(I9_000_Bit09) XIC(I9_000_Bit11) [XIC(I9_000_Bit10) ,XIC(arm1_slc2:1:O.Point_25) ] ]XIO(B14[11].0)[OTE(arm1_slc2:1:O.Point_25) ,OTE(P3) ];
   84: [XIC(arm1_slc2:1:O.Point_26) ,XIC(P4) ]TON(T27[19],?,?);
   85: XIC(arm1_slc2:1:O.Point_25)TON(T27[20],?,?);
   86: XIC(T27[20].DN)XIC(T27[20].EN)XIC(I4_000_Bit02)OTE(arm1_slc2:1:O.Point_26);
   87: XIO(arm1_slc2:1:O.Point_26)XIO(P4)MOV(0.0,F8[100]);
   88: XIC(arm1_slc2:1:O.Point_26)ONS(B3[24].12)MOV(50.0,F8[100]);
